// TIA Portal V18 export
// export: Created 2026-01-09T11:31:55.8642182Z, ExportSetting WithDefaults, DisplayName Totally Integrated Automation Portal, DisplayVersion V18 Update 5, DisplayName TIA Portal Openness, DisplayVersion V18 Update 5, DisplayName TIA Portal Teamcenter Gateway, DisplayVersion V18, DisplayName TIA Portal Version Control Interface, DisplayVersion V18, DisplayName SINAMICS Startdrive Advanced, DisplayVersion V18 SP2 Update 1, DisplayName SINAMICS Startdrive G110M, G120, G120C, G120D, G120P, G115D, DisplayVersion V18 SP2 Update 1, DisplayName SINAMICS Startdrive G130, G150, S120, S150, SINAMICS MV, S210, G220, S200, DisplayVersion V18 SP2 Update 1, DisplayName STEP 7 Professional, DisplayVersion V18 Update 5, DisplayName STEP 7 Safety, DisplayVersion V18, DisplayName WinCC Professional, DisplayVersion V18 Update 5
TagTable "ST350_GengralAnalog"
  STxxx_GeneralAnalogDB_aDev{1} : ST_GeneralAnalog  (PLC tag OP10_GeneralAnalogDB.aDev[1], CPU S71500-2PN_TP700, 1 s)
    TagStructureMember "Common"
      TagStructureMember "nMode"
      TagStructureMember "bEnable"
      TagStructureMember "bError"
      TagStructureMember "bWarning"
      TagStructureMember "bReset"
      TagStructureMember "bDone"
      TagStructureMember "bScreenActive"
      TagStructureMember "nErrorNo"
      TagStructureMember "nWarningNo"
      TagStructureMember "nLastStep"
      TagStructureMember "nCurrentStep"
      TagStructureMember "nNextStep"
      TagStructureMember "tMaxProcessTime"
      TagStructureMember "tActProcessTime"
    TagStructureMember "In"
      TagStructureMember "nActualValueX"
    TagStructureMember "Out"
      TagStructureMember "bReserved"
    TagStructureMember "Para"
      TagStructureMember "General"
        TagStructureMember "rActualValueY"
        TagStructureMember "rSlope"
        TagStructureMember "rConstant"
        TagStructureMember "aPos"
          TagArrayMember "[0]"
            TagStructureMember "nValueX"
            TagStructureMember "nValueY"
          TagArrayMember "[1]"
            TagStructureMember "nValueX"
            TagStructureMember "nValueY"
      TagStructureMember "Set"
        TagStructureMember "rLimitMin"
        TagStructureMember "rLimitMax"
        TagStructureMember "aLimit"
          TagArrayMember "[0]"
            TagStructureMember "rMin"
            TagStructureMember "rMax"
          TagArrayMember "[1]"
            TagStructureMember "rMin"
            TagStructureMember "rMax"
          TagArrayMember "[2]"
            TagStructureMember "rMin"
            TagStructureMember "rMax"
          TagArrayMember "[3]"
            TagStructureMember "rMin"
            TagStructureMember "rMax"
          TagArrayMember "[4]"
            TagStructureMember "rMin"
            TagStructureMember "rMax"
          TagArrayMember "[5]"
            TagStructureMember "rMin"
            TagStructureMember "rMax"
          TagArrayMember "[6]"
            TagStructureMember "rMin"
            TagStructureMember "rMax"
          TagArrayMember "[7]"
            TagStructureMember "rMin"
            TagStructureMember "rMax"
          TagArrayMember "[8]"
            TagStructureMember "rMin"
            TagStructureMember "rMax"
          TagArrayMember "[9]"
            TagStructureMember "rMin"
            TagStructureMember "rMax"
        TagStructureMember "nUnitX"
        TagStructureMember "nUnitY"
      TagStructureMember "Result"
        TagStructureMember "bOk"
        TagStructureMember "bNok"
        TagStructureMember "bOverMin"
        TagStructureMember "bOverMax"
        TagStructureMember "rValueY"
      TagStructureMember "Record"
        TagStructureMember "bClear"
        TagStructureMember "nSetNumber"
        TagStructureMember "nActNumber"
        TagStructureMember "rAverageValueY"
        TagStructureMember "aValueY"
          TagArrayMember "[0]"
          TagArrayMember "[1]"
          TagArrayMember "[2]"
          TagArrayMember "[3]"
          TagArrayMember "[4]"
          TagArrayMember "[5]"
          TagArrayMember "[6]"
          TagArrayMember "[7]"
          TagArrayMember "[8]"
          TagArrayMember "[9]"
          TagArrayMember "[10]"
          TagArrayMember "[11]"
          TagArrayMember "[12]"
          TagArrayMember "[13]"
          TagArrayMember "[14]"
          TagArrayMember "[15]"
          TagArrayMember "[16]"
          TagArrayMember "[17]"
          TagArrayMember "[18]"
          TagArrayMember "[19]"
          TagArrayMember "[20]"
          TagArrayMember "[21]"
          TagArrayMember "[22]"
          TagArrayMember "[23]"
          TagArrayMember "[24]"
          TagArrayMember "[25]"
          TagArrayMember "[26]"
          TagArrayMember "[27]"
          TagArrayMember "[28]"
          TagArrayMember "[29]"
          TagArrayMember "[30]"
          TagArrayMember "[31]"
          TagArrayMember "[32]"
          TagArrayMember "[33]"
          TagArrayMember "[34]"
          TagArrayMember "[35]"
          TagArrayMember "[36]"
          TagArrayMember "[37]"
          TagArrayMember "[38]"
          TagArrayMember "[39]"
          TagArrayMember "[40]"
          TagArrayMember "[41]"
          TagArrayMember "[42]"
          TagArrayMember "[43]"
          TagArrayMember "[44]"
          TagArrayMember "[45]"
          TagArrayMember "[46]"
          TagArrayMember "[47]"
          TagArrayMember "[48]"
          TagArrayMember "[49]"
  STxxx_GeneralAnalogDB_aDev{2} : ST_GeneralAnalog  (PLC tag OP10_GeneralAnalogDB.aDev[2], CPU S71500-2PN_TP700, 1 s)
    TagStructureMember "Common"
      TagStructureMember "nMode"
      TagStructureMember "bEnable"
      TagStructureMember "bError"
      TagStructureMember "bWarning"
      TagStructureMember "bReset"
      TagStructureMember "bDone"
      TagStructureMember "bScreenActive"
      TagStructureMember "nErrorNo"
      TagStructureMember "nWarningNo"
      TagStructureMember "nLastStep"
      TagStructureMember "nCurrentStep"
      TagStructureMember "nNextStep"
      TagStructureMember "tMaxProcessTime"
      TagStructureMember "tActProcessTime"
    TagStructureMember "In"
      TagStructureMember "nActualValueX"
    TagStructureMember "Out"
      TagStructureMember "bReserved"
    TagStructureMember "Para"
      TagStructureMember "General"
        TagStructureMember "rActualValueY"
        TagStructureMember "rSlope"
        TagStructureMember "rConstant"
        TagStructureMember "aPos"
          TagArrayMember "[0]"
            TagStructureMember "nValueX"
            TagStructureMember "nValueY"
          TagArrayMember "[1]"
            TagStructureMember "nValueX"
            TagStructureMember "nValueY"
      TagStructureMember "Set"
        TagStructureMember "rLimitMin"
        TagStructureMember "rLimitMax"
        TagStructureMember "aLimit"
          TagArrayMember "[0]"
            TagStructureMember "rMin"
            TagStructureMember "rMax"
          TagArrayMember "[1]"
            TagStructureMember "rMin"
            TagStructureMember "rMax"
          TagArrayMember "[2]"
            TagStructureMember "rMin"
            TagStructureMember "rMax"
          TagArrayMember "[3]"
            TagStructureMember "rMin"
            TagStructureMember "rMax"
          TagArrayMember "[4]"
            TagStructureMember "rMin"
            TagStructureMember "rMax"
          TagArrayMember "[5]"
            TagStructureMember "rMin"
            TagStructureMember "rMax"
          TagArrayMember "[6]"
            TagStructureMember "rMin"
            TagStructureMember "rMax"
          TagArrayMember "[7]"
            TagStructureMember "rMin"
            TagStructureMember "rMax"
          TagArrayMember "[8]"
            TagStructureMember "rMin"
            TagStructureMember "rMax"
          TagArrayMember "[9]"
            TagStructureMember "rMin"
            TagStructureMember "rMax"
        TagStructureMember "nUnitX"
        TagStructureMember "nUnitY"
      TagStructureMember "Result"
        TagStructureMember "bOk"
        TagStructureMember "bNok"
        TagStructureMember "bOverMin"
        TagStructureMember "bOverMax"
        TagStructureMember "rValueY"
      TagStructureMember "Record"
        TagStructureMember "bClear"
        TagStructureMember "nSetNumber"
        TagStructureMember "nActNumber"
        TagStructureMember "rAverageValueY"
        TagStructureMember "aValueY"
          TagArrayMember "[0]"
          TagArrayMember "[1]"
          TagArrayMember "[2]"
          TagArrayMember "[3]"
          TagArrayMember "[4]"
          TagArrayMember "[5]"
          TagArrayMember "[6]"
          TagArrayMember "[7]"
          TagArrayMember "[8]"
          TagArrayMember "[9]"
          TagArrayMember "[10]"
          TagArrayMember "[11]"
          TagArrayMember "[12]"
          TagArrayMember "[13]"
          TagArrayMember "[14]"
          TagArrayMember "[15]"
          TagArrayMember "[16]"
          TagArrayMember "[17]"
          TagArrayMember "[18]"
          TagArrayMember "[19]"
          TagArrayMember "[20]"
          TagArrayMember "[21]"
          TagArrayMember "[22]"
          TagArrayMember "[23]"
          TagArrayMember "[24]"
          TagArrayMember "[25]"
          TagArrayMember "[26]"
          TagArrayMember "[27]"
          TagArrayMember "[28]"
          TagArrayMember "[29]"
          TagArrayMember "[30]"
          TagArrayMember "[31]"
          TagArrayMember "[32]"
          TagArrayMember "[33]"
          TagArrayMember "[34]"
          TagArrayMember "[35]"
          TagArrayMember "[36]"
          TagArrayMember "[37]"
          TagArrayMember "[38]"
          TagArrayMember "[39]"
          TagArrayMember "[40]"
          TagArrayMember "[41]"
          TagArrayMember "[42]"
          TagArrayMember "[43]"
          TagArrayMember "[44]"
          TagArrayMember "[45]"
          TagArrayMember "[46]"
          TagArrayMember "[47]"
          TagArrayMember "[48]"
          TagArrayMember "[49]"
